# EPICS autosave request: iocBoot/obsolete/ioc13esp_test/auto_settings.req
file "CARS_motor_settings.req",         P=$(P), M=m1
file "CARS_motor_settings.req",         P=$(P), M=m2
file "CARS_motor_settings.req",         P=$(P), M=m3
